INTERFACE PUBLIC StoppingCommands

METHOD PUBLIC StateComplete
END_METHOD

END_INTERFACE

(* stored: Version 1.1.0.1, ProductVersion 3.1.4026.12
   Itf StoppingCommands: Id {28886706-ab5d-0d83-1519-135622573c5d}
   Method StateComplete: Id {039fc134-3968-456c-a60f-00bf64667845} *)
